(* IEC 61131-3 sources: JaccoSigma/tempclass/Class/_CanOpenSDOTab, 1 file *)

(* ---- _CanOpenSDOTab.st ---- *)
(*!
<Class
	Name               = "_CanOpenSDOTab"
	Revision           = "1.0"
	RealtimeTask       = "false"
	CyclicTask         = "false"
	BackgroundTask     = "false"
	Sigmatek           = "true"
	OSInterface        = "false"
	HighPriority       = "false"
	Automatic          = "false"
	UpdateMode         = "Prescan"
	IconPath           = ".\Class\_CanOpenSDOTab\Drive1.ico"
	SharedCommandTable = "true"
	Objectsize         = "(382,120)"
	Comment            = "Call provides SDO Parameter-Table.&#13;&#10;Must be overwritten by User, because default Table is empty!">
	<Channels>
		<Server Name="ClassSvr" Visualized="false" Initialize="false" WriteProtected="true" Retentive="false"/>
	</Channels>
	<RevDoku>
		<Owner Company="Sigmatek" Author="WesAnd"/>
		<Dokumentation Revision="1.0" Date="08.08.2012" Author="WesAnd" Company="Sigmatek" Description="Initial Version"/>
	</RevDoku>
</Class>
*)
_CanOpenSDOTab : CLASS
  //Servers:
	ClassSvr 	: SvrChCmd_DINT;
  //Clients:
  //Variables:
  //Functions:
				//! <Function Comment="Methode is called from class _CanOpenBasic to get Pointer to SDO-Parametertable." Name="GetTabPtr"/>
	FUNCTION VIRTUAL GLOBAL GetTabPtr
		VAR_OUTPUT
			dTabPtr 	: DINT;			//! <Variable Comment="Pointer to SDO-Parametertable.&#13;&#10;Format: Index (2 Byte), SubIndex (1 Byte), Data (4 Byte), Length (1 Byte)." Name="GetTabPtr.dTabPtr"/>
		END_VAR;

	FUNCTION TAB ParaTab;
  //Tables:
	FUNCTION @STD
		VAR_OUTPUT
			ret_code	: CONFSTATES;
		END_VAR;
	FUNCTION GLOBAL TAB @CT_;
END_CLASS;

FUNCTION VIRTUAL GLOBAL _CanOpenSDOTab::GetTabPtr
	VAR_OUTPUT
		dTabPtr 	: DINT;
	END_VAR

  //Return Pointer to Table
  dTabptr := (#ParaTab())$DINT;

END_FUNCTION

FUNCTION TAB _CanOpenSDOTab::ParaTab

  // INDEX(2Byte)   SUBINDEX(1Byte)   DATA(4Byte)   LENGTH(1Byte)
  16#200A$INT,      16#02$USINT,      3$DINT,       2$USINT,      // Set Accesslevel for CanOpen to 3

END_FUNCTION
